                    bPartRemovedConfirmedForExchange := FALSE;

                    eOperatorExchangeState :=
                        E_OperatorExchangeState.ExchangeComplete;

                ELSE

                    // Original enabled Puck Locker sequence.
                    eOperatorExchangeState :=
                        E_OperatorExchangeState.WaitingForPuckRemoval;

                END_IF


            // -------------------------------------------------------------
            // FAIL result.
            // -------------------------------------------------------------
            ELSIF bPendingOperatorResultFail THEN

                // The rejected part must be placed at the reject sensor.
                eOperatorExchangeState :=
                    E_OperatorExchangeState.WaitingForRejectConfirmation;

            END_IF

        END_IF


    // ========================================================================
    E_OperatorExchangeState.WaitingForPuckRemoval:
    // ========================================================================

        bOperatorExchangeComplete := FALSE;


        // Recovery protection:
        //
        // If the Puck Locker is disabled while the sequence is already in
        // this state, no puck removal must be awaited.
        IF GVL_HMI.stPuckLocker.eMode =
            E_PuckLockerMode.Disabled THEN

            bPartRemovedConfirmedForExchange := FALSE;

            eOperatorExchangeState :=
                E_OperatorExchangeState.ExchangeComplete;

        ELSE

            // Once the locker accepts the release request,
            // the part-removal handshake is no longer needed.
            IF GVL_MASTER.stPuckLocker.eState =
                E_PuckLockerState.ReleasingPuck THEN

                bPartRemovedConfirmedForExchange := FALSE;

            END_IF


            // Advance when the old puck is physically gone.
            //
            // Do not require the locker to remain in ReleasingPuck.
            IF NOT GVL_MASTER.stPuckLocker.bPuckDetected THEN

                eOperatorExchangeState :=
                    E_OperatorExchangeState.WaitingForNewPuck;

            END_IF

        END_IF


    // ========================================================================
    E_OperatorExchangeState.WaitingForRejectConfirmation:
    // ========================================================================

        bOperatorExchangeComplete := FALSE;


        // Latch the reject-bin sensor pulse.
        IF rtPartPresentReject.Q THEN

            bRejectConfirmedForExchange := TRUE;

        END_IF


        // Complete the rejected-part exchange when:
        //
        // 1. The rejected part has been confirmed at the reject sensor.
        // 2. The part is no longer present in the operator nest.
        // 3. The Puck Locker is disabled, or the puck remains present
        //    and locked.
        IF bRejectConfirmedForExchange
			   AND bPartRemovedConfirmedForExchange
			   AND
			   (
                GVL_HMI.stPuckLocker.eMode =
                    E_PuckLockerMode.Disabled

                OR
                (
                    GVL_MASTER.stPuckLocker.bPuckDetected
                    AND
                    GVL_MASTER.stPuckLocker.bPuckLocked
                    AND
                    GVL_MASTER.stPuckLocker.eState =
                        E_PuckLockerState.Locked
                )
           ) THEN

            bPartRemovedConfirmedForExchange := FALSE;

            eOperatorExchangeState :=
                E_OperatorExchangeState.ExchangeComplete;

        END_IF


    // ========================================================================
    E_OperatorExchangeState.WaitingForNewPuck:
    // ========================================================================

        bOperatorExchangeComplete := FALSE;


        // Recovery protection:
        //
        // A replacement puck is not required when the locker is disabled.
        IF GVL_HMI.stPuckLocker.eMode =
            E_PuckLockerMode.Disabled THEN

            eOperatorExchangeState :=
                E_OperatorExchangeState.ExchangeComplete;


        // Original enabled Puck Locker sequence.
        ELSIF GVL_MASTER.stPuckLocker.bPuckDetected THEN

            eOperatorExchangeState :=
                E_OperatorExchangeState.WaitingForPuckLocked;

        END_IF


    // ========================================================================
    E_OperatorExchangeState.WaitingForPuckLocked:
    // ========================================================================

        bOperatorExchangeComplete := FALSE;


        // Recovery protection:
        //
        // Physical puck locking is not required when the locker is disabled.
        IF GVL_HMI.stPuckLocker.eMode =
            E_PuckLockerMode.Disabled THEN

            eOperatorExchangeState :=
                E_OperatorExchangeState.ExchangeComplete;


        // Original enabled Puck Locker sequence.
        ELSIF GVL_MASTER.stPuckLocker.bPuckDetected
           AND GVL_MASTER.stPuckLocker.bPuckLocked
           AND GVL_MASTER.stPuckLocker.eState =
                E_PuckLockerState.Locked THEN

            // Loading a new part remains optional.
            eOperatorExchangeState :=
                E_OperatorExchangeState.ExchangeComplete;

        END_IF


    // ========================================================================
    E_OperatorExchangeState.WaitingForPartLoading:
    // ========================================================================

        // Original behavior preserved.
        //
        // Require an actual OFF -> ON transition from the operator nest
        // sensor. The puck must also be present and locked.
        IF GVL_MASTER.astNestTracking[
                iOperatorNestIndex
           ].bPartLoadedPulse
           AND GVL_MASTER.stPuckLocker.bPuckDetected
           AND GVL_MASTER.stPuckLocker.bPuckLocked
           AND GVL_MASTER.stPuckLocker.eState =
                E_PuckLockerState.Locked THEN

            eOperatorExchangeState :=
                E_OperatorExchangeState.ExchangeComplete;

        END_IF


    // ========================================================================
    E_OperatorExchangeState.ExchangeComplete:
    // ========================================================================

        // Keep the index permission active until the table starts moving.
        bOperatorExchangeComplete := TRUE;


        // The previous result and its disposition are complete.
        M_ClearCompletedOperatorNestResult();


        IF GVL_MASTER.stNestTable.bNestInMotion THEN

            bPendingOperatorResultPass := FALSE;
            bPendingOperatorResultFail := FALSE;

            bPartRemovedConfirmedForExchange := FALSE;
            bRejectConfirmedForExchange := FALSE;

            eOperatorExchangeState :=
                E_OperatorExchangeState.WaitingForTableIndexComplete;

        END_IF


    // ========================================================================
    E_OperatorExchangeState.WaitingForTableIndexComplete:
    // ========================================================================

        bOperatorExchangeComplete := TRUE;


        IF eNestState = E_NestState.TESTING
           AND NOT GVL_MASTER.stNestTable.bNestInMotion
           AND GVL_MASTER.stNestTable.bNestReadySensor
           AND GVL_MASTER.stNestTable.bNestLockedSensor
           AND eCurrentNestPos <> E_NestPosition.Unknown THEN

            bOperatorExchangeComplete := FALSE;

            bPendingOperatorResultPass := FALSE;
            bPendingOperatorResultFail := FALSE;

            bPartRemovedConfirmedForExchange := FALSE;
            bRejectConfirmedForExchange := FALSE;

            eOperatorExchangeState :=
                E_OperatorExchangeState.Idle;

        END_IF


    // ========================================================================
    ELSE
    // ========================================================================

        bOperatorExchangeComplete := FALSE;

        bPendingOperatorResultPass := FALSE;
        bPendingOperatorResultFail := FALSE;

        bPartRemovedConfirmedForExchange := FALSE;
        bRejectConfirmedForExchange := FALSE;

        eOperatorExchangeState :=
            E_OperatorExchangeState.Idle;

END_CASE
END_METHOD

METHOD PRIVATE M_PreExecution : BOOL
VAR

END_VAR
// =================================================================================
// SYSTEM TIMERS
// =================================================================================
// Update initialization and safety timers on every PLC scan cycle
tonSys_Init(IN := GVL_MASTER.stMachineStatus.bInitialising);
tonSys_InitTimeout(IN := GVL_MASTER.stMachineStatus.bInitialising);

// TwinSAFE circuit stabilization timer (10 seconds)
tonSafety(IN := (GVL_MASTER.stMachineStatus.eMachineState = E_MachineState.SAFETY), PT := T#10S);

// 
//  fbStopTrigger(CLK := GVL_Master.i_bButtonStop);
//  bButtonStop := fbStopTrigger.Q;

// =================================================================================
// HMI MESSAGE CLEARING
// =================================================================================
// Clear old system messages if the machine is not actively in production
// Uses the proper ENUM namespace from your MASTER folder
IF GVL_MASTER.stMachineStatus.eMachineState <> E_MachineState.SYSTEM_AUTO_CYCLE THEN
    sMachineMessage := '';            
END_IF


// =================================================================================
// CRITICAL FAULT INTERLOCK (Watchdog)
// =================================================================================
// If Kistler hardware is NOT ready, force the state machine to FAULT immediately
// Exception: Do not override if the system is currently in SAFETY or POWER_UP
IF NOT GVL_MASTER.bKistlerSystemReady 
    AND GVL_MASTER.stMachineStatus.eMachineState <> E_MachineState.SAFETY 
    AND GVL_MASTER.stMachineStatus.eMachineState <> E_MachineState.SYSTEM_POWER_UP THEN
    
    GVL_MASTER.stMachineStatus.eMachineState := E_MachineState.FAULT;
END_IF


// =================================================================================
// START LEDs BUTTON OFF
// =================================================================================
eMode_LED_Start := E_LEDs_Mode.OFF;
eMode_LED_Reset := E_LEDs_Mode.OFF;

// =================================================================================
// METHOD EXECUTION FEEDBACK (Return True)
// =================================================================================
// Returning TRUE confirms the pre-execution routine completed successfully
M_PreExecution := TRUE;
END_METHOD

METHOD M_ProcessCycle : BOOL
VAR
bControlledStopActive 	: BOOL;
rTrigTwoHands : R_TRIG; // Edge trigger to detect single press of the two-hand safety signal

bManualIndexerOnly        : BOOL;
bManualKistlerOnly        : BOOL;
bManualIndexerAndKistler  : BOOL;



END_VAR
// Process cycle is allowed during:
//
// 1. Automatic production.
// 2. Manual Mode when the Kistler or indexer manual function is enabled.
bProcessCycleAllowed :=
    (
        GVL_MASTER.stMachineStatus.eMachineState =
            E_MachineState.SYSTEM_AUTO_CYCLE
    )
    OR
    (
        GVL_MASTER.stMachineStatus.eMachineState =
            E_MachineState.MANUAL_MODE

        AND
        (
            GVL_HMI.i_bHMIKistlerManualEnable
            OR
            GVL_HMI.i_bHMIIndexerManualEnable
        )
    );


bManualIndexerOnly :=
    GVL_HMI.i_bHMIIndexerManualEnable
    AND NOT GVL_HMI.i_bHMIKistlerManualEnable;


bManualKistlerOnly :=
    GVL_HMI.i_bHMIKistlerManualEnable
    AND NOT GVL_HMI.i_bHMIIndexerManualEnable;


bManualIndexerAndKistler :=
    GVL_HMI.i_bHMIIndexerManualEnable
    AND GVL_HMI.i_bHMIKistlerManualEnable;


// -----------------------------------------------------------------------------
// If process execution is not permitted, reset the temporary process states.
//
// Stored nest PASS/FAIL results must not be cleared by M_ResetProcessCycle.
// -----------------------------------------------------------------------------
IF NOT bProcessCycleAllowed THEN

    M_ResetProcessCycle();

    RETURN;

END_IF


// -----------------------------------------------------------------------------
// Common timers and edge detections.
// -----------------------------------------------------------------------------
rTrigTwoHands(
    CLK := GVL_IO.stSafety.bTwoHandsSafe
);


tTwoHandTargetTime :=
    REAL_TO_TIME(rHmiTwoHandPresetTime);


tTwoHandHoldTimer(
    IN := GVL_IO.stSafety.bTwoHandsSafe,
    PT := tTwoHandTargetTime
);


rtPartPresentReject(
    CLK := GVL_MASTER.stSensors.bPartPresent_Reject
);


// ============================================================================
// COMMON POSITION AND TRACKING UPDATE
//
// These methods are required in both Auto and Manual Mode.
// ============================================================================
eCurrentNestPos :=
    M_GetCurrentPosition();


M_UpdateActiveNestPositions();

M_UpdateOperatorNestTracking();


// ============================================================================
// AUTOMATIC OPERATOR EXCHANGE
//
// The following methods belong only to automatic production.
//
// They must not:
//
// - send a PASS/FAIL disposition while in Manual Mode;
// - release a puck during Manual Mode;
// - clear a completed nest result during Manual Mode;
// - block manual index movement waiting for part removal;
// - block manual index movement waiting for reject confirmation;
// - block manual index movement waiting for a puck.
// ============================================================================
IF GVL_MASTER.stMachineStatus.eMachineState =
    E_MachineState.SYSTEM_AUTO_CYCLE THEN

    M_UpdatePuckLockerPartRemovalStatus();

    M_ConfirmPuckLockerDisposition();

    M_PuckLockerDisposition();

    M_OperatorExchangeControl();

ELSE

    // Prevent a stale removal confirmation from being sent to the
    // Puck Locker while the machine is operating manually.
    GVL_MASTER.stPuckLocker.bPartRemovedFromNest := FALSE;

END_IF


// -----------------------------------------------------------------------------
// Determine whether the current physical table position is different from
// the most recently processed Kistler position.
// -----------------------------------------------------------------------------
bNestNewPositionReady :=
    (
        eCurrentNestPos <> E_NestPosition.UNKNOWN
    )
    AND
    (
        eCurrentNestPos <> eLastTestedNestPos
    );


// -----------------------------------------------------------------------------
// Capture live Kistler values while an automatic or manual sequence is active.
//
// This does not store PASS/FAIL. It only updates the live maximum values.
// -----------------------------------------------------------------------------
IF GVL_MASTER.stProcess.bKistlerCycleRequest
   AND NOT stKistlerOutTelegram.bSequenceEnd THEN

    M_HMIKistlerResult(
        eNestPosition := eCurrentNestPos,
        bPartOK       := FALSE,
        bPartNOK      := FALSE,
        rForce        := stKistler_Status.rLiveForce,
        rDistance     := stKistler_Status.rLiveDistance,
        bResetValues  := FALSE
    );

END_IF


// ============================================================================
// PROCESS CYCLE COORDINATOR
// ============================================================================
CASE GVL_MASTER.stMachineStatus.eMachineState OF


    // ========================================================================
    // AUTOMATIC CYCLE
    // ========================================================================
    E_MachineState.SYSTEM_AUTO_CYCLE:

        CASE eProcessCycleState OF


            // =================================================================
            E_ProcessCycle_State.IDLE:
            // =================================================================

                GVL_MASTER.stProcess.bKistlerCycleRequest := FALSE;
                GVL_MASTER.stProcess.bKistlerCycleDone    := FALSE;
                GVL_MASTER.stProcess.bKistlerHomeDone     := FALSE;
                GVL_MASTER.stProcess.bReleaseNestRotation := FALSE;

                tonAfterKistlerDelay(IN := FALSE);

                IF bProcessCycleAllowed THEN

                    eProcessCycleState :=
                        E_ProcessCycle_State.WAIT_NEST_TESTING_READY;

                END_IF


            // =================================================================
            E_ProcessCycle_State.WAIT_NEST_TESTING_READY:
            // =================================================================

                GVL_MASTER.stProcess.bKistlerCycleRequest := FALSE;
                GVL_MASTER.stProcess.bReleaseNestRotation := FALSE;

                tonAfterKistlerDelay(IN := FALSE);


                IF NOT bProcessCycleAllowed THEN

                    eProcessCycleState :=
                        E_ProcessCycle_State.IDLE;


                // -------------------------------------------------------------
                // Invalid table position.
                //
                // Never execute the Kistler if the PLC cannot determine which
                // physical nest is currently at the test station.
                // -------------------------------------------------------------
                ELSIF GVL_MASTER.stProcess.bNestTestingReady
                      AND eNestState = E_NestState.TESTING
                      AND eCurrentNestPos =
                            E_NestPosition.UNKNOWN THEN

                    GVL_MASTER.stProcess.bKistlerCycleRequest := FALSE;
                    GVL_MASTER.stProcess.bReleaseNestRotation := FALSE;
                    GVL_MASTER.stProcess.bKistlerCycleDone    := FALSE;
                    GVL_MASTER.stProcess.bKistlerHomeDone     := FALSE;

                    eProcessCycleState :=
                        E_ProcessCycle_State.FAULT;


                // -------------------------------------------------------------
                // Same position already processed, or no part at Kistler.
                //
                // Do not execute another Kistler cycle. Release the table.
                // -------------------------------------------------------------
                ELSIF GVL_MASTER.stProcess.bNestTestingReady
                      AND eNestState = E_NestState.TESTING
                      AND GVL_MASTER.stNestTable.bNestReadySensor
                      AND GVL_MASTER.stNestTable.bNestLockedSensor
                      AND NOT GVL_MASTER.stNestTable.bNestInMotion
                      AND eCurrentNestPos <>
                            E_NestPosition.UNKNOWN
                      AND
                      (
                          NOT bNestNewPositionReady
                          OR
                          NOT GVL_MASTER.stSensors.bPartPresent_Kistler
                      ) THEN

                    GVL_MASTER.stProcess.bKistlerCycleRequest := FALSE;
                    GVL_MASTER.stProcess.bKistlerCycleDone    := FALSE;

                    // Kistler side is considered complete because there is
                    // no valid new part to test.
                    GVL_MASTER.stProcess.bKistlerHomeDone := TRUE;


                    IF bNestNewPositionReady THEN

                        // New position without a part.
                        // Remove any previous HMI measurement result.
                        M_HMIKistlerResult(
                            eNestPosition := eCurrentNestPos,
                            bPartOK       := FALSE,
                            bPartNOK      := FALSE,
                            rForce        := 0.0,
                            rDistance     := 0.0,
                            bResetValues  := TRUE
                        );

                        eLastTestedNestPos :=
                            eCurrentNestPos;

                    END_IF


                    GVL_MASTER.stProcess.bReleaseNestRotation := TRUE;

                    eProcessCycleState :=
                        E_ProcessCycle_State.RELEASE_NEST;


                // -------------------------------------------------------------
                // New enabled nest containing a part.
                //
                // Execute the Kistler sequence.
                // -------------------------------------------------------------
                ELSIF GVL_MASTER.stProcess.bNestTestingReady
                      AND eNestState = E_NestState.TESTING
                      AND GVL_MASTER.stNestTable.bNestReadySensor
                      AND GVL_MASTER.stNestTable.bNestLockedSensor
                      AND NOT GVL_MASTER.stNestTable.bNestInMotion
                      AND stKistler_Status.eKistlerState =
                            E_KistlerState.READY
                      AND NOT stKistler_Status.bError
                      AND NOT bKistlerRecoveryHomeRequest
                      AND bNestNewPositionReady
                      AND GVL_MASTER.stSensors.bPartPresent_Kistler
                      AND M_IsNestEnabled(eCurrentNestPos) THEN

                    GVL_MASTER.stProcess.bKistlerCycleDone := FALSE;
                    GVL_MASTER.stProcess.bKistlerHomeDone  := FALSE;

                    bKistlerResultStored := FALSE;


                    // Clear the previous HMI measurement values.
                    M_HMIKistlerResult(
                        eNestPosition := eCurrentNestPos,
                        bPartOK       := FALSE,
                        bPartNOK      := FALSE,
                        rForce        := 0.0,
                        rDistance     := 0.0,
                        bResetValues  := TRUE
                    );


                    eProcessCycleState :=
                        E_ProcessCycle_State.REQUEST_KISTLER;


                // -------------------------------------------------------------
                // Nest disabled from HMI.
                //
                // Skip the Kistler test and release the table normally.
                // -------------------------------------------------------------
                ELSIF GVL_MASTER.stProcess.bNestTestingReady
                      AND eNestState = E_NestState.TESTING
                      AND GVL_MASTER.stNestTable.bNestReadySensor
                      AND GVL_MASTER.stNestTable.bNestLockedSensor
                      AND NOT GVL_MASTER.stNestTable.bNestInMotion
                      AND eCurrentNestPos <>
                            E_NestPosition.UNKNOWN
                      AND bNestNewPositionReady
                      AND GVL_MASTER.stSensors.bPartPresent_Kistler
                      AND NOT M_IsNestEnabled(eCurrentNestPos) THEN

                    GVL_MASTER.stProcess.bKistlerCycleRequest := FALSE;
                    GVL_MASTER.stProcess.bKistlerCycleDone    := FALSE;
                    GVL_MASTER.stProcess.bKistlerHomeDone     := TRUE;


                    M_HMIKistlerResult(
                        eNestPosition := eCurrentNestPos,
                        bPartOK       := FALSE,
                        bPartNOK      := FALSE,
                        rForce        := 0.0,
                        rDistance     := 0.0,
                        bResetValues  := TRUE
                    );


                    eLastTestedNestPos :=
                        eCurrentNestPos;

                    GVL_MASTER.stProcess.bReleaseNestRotation :=
                        TRUE;

                    eProcessCycleState :=
                        E_ProcessCycle_State.RELEASE_NEST;

                END_IF


            // =================================================================
            E_ProcessCycle_State.REQUEST_KISTLER:
            // =================================================================

                GVL_MASTER.stProcess.bKistlerCycleRequest := TRUE;


                IF stKistler_Status.bError THEN

                    GVL_MASTER.stProcess.bKistlerCycleRequest :=
                        FALSE;

                    eProcessCycleState :=
                        E_ProcessCycle_State.FAULT;


                ELSIF stKistler_Status.eKistlerState <>
                      E_KistlerState.READY THEN

                    eProcessCycleState :=
                        E_ProcessCycle_State.WAIT_KISTLER_DONE;

                END_IF


            // =================================================================
            E_ProcessCycle_State.WAIT_KISTLER_DONE:
            // =================================================================

                // Keep the request active while the Kistler is executing.
                GVL_MASTER.stProcess.bKistlerCycleRequest := TRUE;


                IF stKistler_Status.bError THEN

                    GVL_MASTER.stProcess.bKistlerCycleRequest :=
                        FALSE;

                    eProcessCycleState :=
                        E_ProcessCycle_State.FAULT;


                ELSIF stKistler_Status.eKistlerState =
                      E_KistlerState.DONE THEN

                    GVL_MASTER.stProcess.bKistlerCycleRequest :=
                        FALSE;

                    GVL_MASTER.stProcess.bKistlerCycleDone :=
                        TRUE;

                    eProcessCycleState :=
                        E_ProcessCycle_State.WAIT_KISTLER_HOME;

                END_IF


            // =================================================================
            E_ProcessCycle_State.WAIT_KISTLER_HOME:
            // =================================================================

                M_StoreKistlerResult();

                GVL_MASTER.stProcess.bKistlerCycleRequest := FALSE;


                IF stKistler_Status.bError THEN

                    eProcessCycleState :=
                        E_ProcessCycle_State.FAULT;


                ELSIF stKistlerOutTelegram.bHomePosReached
                      OR stKistlerOutTelegram.bRefPosReached
                      OR stKistler_Status.bInPosition THEN

                    GVL_MASTER.test :=
                        GVL_MASTER.test + 1;

                    GVL_MASTER.stProcess.bKistlerHomeDone :=
                        TRUE;

                    GVL_MASTER.stProcess.bKistlerCycleDone :=
                        TRUE;


                    // ---------------------------------------------------------
                    // Store the process result.
                    // ---------------------------------------------------------
                    IF stKistler_Status.bPartOK THEN

                        GVL_MASTER.stProcess.bKistlerResultOK :=
                            TRUE;

                        GVL_MASTER.stProcess.bKistlerResultNOK :=
                            FALSE;


                    ELSIF stKistler_Status.bPartNOK THEN

                        GVL_MASTER.stProcess.bKistlerResultOK :=
                            FALSE;

                        GVL_MASTER.stProcess.bKistlerResultNOK :=
                            TRUE;


                    ELSE

                        // Test ended without a valid OK/NOK result.
                        // Preserve the existing behavior.
                        RETURN;

                    END_IF


                    eLastTestedNestPos :=
                        eCurrentNestPos;


                    IF NOT M_HMIKistlerResult(
                        eNestPosition := eCurrentNestPos,
                        bPartOK       := stKistler_Status.bPartOK,
                        bPartNOK      := stKistler_Status.bPartNOK,
                        rForce        := stKistler_Status.rLiveForce,
                        rDistance     := stKistler_Status.rLiveDistance,
                        bResetValues  := FALSE
                    ) THEN

                        RETURN;

                    END_IF


                    eProcessCycleState :=
                        E_ProcessCycle_State.WAIT_AFTER_KISTLER;

                END_IF


            // =================================================================
            E_ProcessCycle_State.WAIT_AFTER_KISTLER:
            // =================================================================

                IF stKistlerOutTelegram.bSequenceEnd
                   AND
                   (
                       stKistlerOutTelegram.bHomePosReached
                       OR
                       stKistlerOutTelegram.bRefPosReached
                       OR
                       stKistler_Status.bInPosition
                   ) THEN

                    GVL_MASTER.stProcess.bReleaseNestRotation :=
                        TRUE;

                    eProcessCycleState :=
                        E_ProcessCycle_State.RELEASE_NEST;

                END_IF


            // =================================================================
            E_ProcessCycle_State.RELEASE_NEST:
            // =================================================================

                // Keep the release request active until NestTableControl
                // consumes it.
                GVL_MASTER.stProcess.bReleaseNestRotation := TRUE;


                IF eNestState <> E_NestState.TESTING
                   OR NOT GVL_MASTER.stProcess.bNestTestingReady THEN

                    GVL_MASTER.stProcess.bReleaseNestRotation :=
                        FALSE;

                    GVL_MASTER.stProcess.bKistlerCycleRequest :=
                        FALSE;

                    GVL_MASTER.stProcess.bKistlerCycleDone :=
                        FALSE;

                    GVL_MASTER.stProcess.bKistlerHomeDone :=
                        FALSE;

                    tonAfterKistlerDelay(IN := FALSE);


                    eProcessCycleState :=
                        E_ProcessCycle_State.WAIT_NEST_TESTING_READY;

                END_IF


            // =================================================================
            E_ProcessCycle_State.FAULT:
            // =================================================================

                GVL_MASTER.stProcess.bKistlerCycleRequest := FALSE;
                GVL_MASTER.stProcess.bReleaseNestRotation := FALSE;

                tonAfterKistlerDelay(IN := FALSE);

                M_ResetProcessCycle();

                GVL_MASTER.stMachineStatus.eMachineState :=
                    E_MachineState.FAULT;


                IF GVL_MASTER.stMachineStatus.bStopped THEN

                    eProcessCycleState :=
                        E_ProcessCycle_State.IDLE;

                END_IF


            // =================================================================
            ELSE
            // =================================================================

                eProcessCycleState :=
                    E_ProcessCycle_State.IDLE;

        END_CASE


    // ========================================================================
    // MANUAL MODE
    // ========================================================================
    E_MachineState.MANUAL_MODE:

        CASE eProcessCycleState OF


            // =================================================================
            E_ProcessCycle_State.IDLE:
            // =================================================================

                GVL_MASTER.stProcess.bKistlerCycleRequest := FALSE;
                GVL_MASTER.stProcess.bKistlerCycleDone    := FALSE;
                GVL_MASTER.stProcess.bKistlerHomeDone     := FALSE;
                GVL_MASTER.stProcess.bReleaseNestRotation := FALSE;

                GVL_MASTER.stProcess.bKistlerResultOK  := FALSE;
                GVL_MASTER.stProcess.bKistlerResultNOK := FALSE;

                tonAfterKistlerDelay(IN := FALSE);


                IF bManualIndexerOnly
                   OR bManualIndexerAndKistler THEN

                    eProcessCycleState :=
                        E_ProcessCycle_State.WAIT_NEST_TESTING_READY;


                ELSIF bManualKistlerOnly
                      AND NOT GVL_MASTER.stProcess.bNestTestingReady
                      AND stKistler_Status.eKistlerState =
                            E_KistlerState.READY
                      AND NOT stKistler_Status.bError
                      AND NOT bKistlerRecoveryHomeRequest THEN

                    GVL_MASTER.stProcess.bNestTestingReady :=
                        FALSE;

                    eProcessCycleState :=
                        E_ProcessCycle_State.REQUEST_KISTLER;

                END_IF


            // =================================================================
            E_ProcessCycle_State.WAIT_NEST_TESTING_READY:
            // =================================================================

                GVL_MASTER.stProcess.bKistlerCycleRequest := FALSE;
                GVL_MASTER.stProcess.bReleaseNestRotation := FALSE;

                tonAfterKistlerDelay(IN := FALSE);


                IF NOT (
                    bManualIndexerOnly
                    OR bManualIndexerAndKistler
                ) THEN

                    eProcessCycleState :=
                        E_ProcessCycle_State.IDLE;


                ELSIF GVL_MASTER.stProcess.bNestTestingReady
                      AND eNestState = E_NestState.TESTING
                      AND bManualIndexerAndKistler
                      AND stKistler_Status.eKistlerState =
                            E_KistlerState.READY
                      AND NOT stKistler_Status.bError
                      AND NOT bKistlerRecoveryHomeRequest THEN

                    eProcessCycleState :=
                        E_ProcessCycle_State.REQUEST_KISTLER;


                ELSIF GVL_MASTER.stProcess.bNestTestingReady
                      AND eNestState = E_NestState.TESTING
                      AND bManualIndexerOnly THEN

                    GVL_MASTER.stProcess.bKistlerCycleRequest :=
                        FALSE;

                    GVL_MASTER.stProcess.bKistlerHomeDone :=
                        TRUE;

                    GVL_MASTER.stProcess.bReleaseNestRotation :=
                        TRUE;

                    eProcessCycleState :=
                        E_ProcessCycle_State.RELEASE_NEST;

                END_IF


            // =================================================================
            E_ProcessCycle_State.REQUEST_KISTLER:
            // =================================================================

                // Kistler already reacted.
                IF stKistler_Status.eKistlerState <>
                    E_KistlerState.READY THEN

                    eProcessCycleState :=
                        E_ProcessCycle_State.WAIT_KISTLER_DONE;


                // -------------------------------------------------------------
                // Manual Kistler only.
                //
                // Start only on the two-hand rising edge.
                // -------------------------------------------------------------
                ELSIF bManualKistlerOnly
                      AND GVL_IO.stSafety.bSafetyOK
                      AND rTrigTwoHands.Q
                      AND GVL_MASTER.stNestTable.bNestReadySensor
                      AND GVL_MASTER.stNestTable.bNestLockedSensor
                      AND NOT stKistler_Status.bError
                      AND NOT bKistlerRecoveryHomeRequest THEN

                    GVL_MASTER.stProcess.bKistlerCycleRequest :=
                        TRUE;


                // -------------------------------------------------------------
                // Manual indexer and Kistler.
                // -------------------------------------------------------------
                ELSIF bManualIndexerAndKistler
                      AND GVL_MASTER.stProcess.bNestTestingReady
                      AND eNestState = E_NestState.TESTING
                      AND GVL_MASTER.stNestTable.bNestReadySensor
                      AND GVL_MASTER.stNestTable.bNestLockedSensor
                      AND NOT GVL_MASTER.stNestTable.bNestInMotion
                      AND eCurrentNestPos <>
                            E_NestPosition.UNKNOWN
                      AND bNestNewPositionReady
                      AND NOT stKistler_Status.bError
                      AND NOT bKistlerRecoveryHomeRequest THEN

                    GVL_MASTER.stProcess.bKistlerCycleRequest :=
                        TRUE;


                ELSIF stKistler_Status.bError THEN

                    GVL_MASTER.stProcess.bKistlerCycleRequest :=
                        FALSE;

                    eProcessCycleState :=
                        E_ProcessCycle_State.FAULT;

                END_IF


            // =================================================================
            E_ProcessCycle_State.WAIT_KISTLER_DONE:
            // =================================================================

                GVL_MASTER.stProcess.bKistlerCycleRequest := TRUE;


                IF stKistler_Status.bError THEN

                    GVL_MASTER.stProcess.bKistlerCycleRequest :=
                        FALSE;

                    eProcessCycleState :=
                        E_ProcessCycle_State.FAULT;


                ELSIF stKistler_Status.eKistlerState =
                      E_KistlerState.DONE THEN

                    // Capture the final available measurements.
                    M_HMIKistlerResult(
                        eNestPosition := eCurrentNestPos,
                        bPartOK       := FALSE,
                        bPartNOK      := FALSE,
                        rForce        := stKistler_Status.rLiveForce,
                        rDistance     := stKistler_Status.rLiveDistance,
                        bResetValues  := FALSE
                    );


                    GVL_MASTER.stProcess.bKistlerCycleRequest :=
                        FALSE;

                    GVL_MASTER.stProcess.bKistlerCycleDone :=
                        TRUE;


                    IF bManualIndexerAndKistler THEN

                        eLastTestedNestPos :=
                            eCurrentNestPos;

                        eProcessCycleState :=
                            E_ProcessCycle_State.WAIT_KISTLER_HOME;

                    ELSE

                        eProcessCycleState :=
                            E_ProcessCycle_State.IDLE;

                    END_IF

                END_IF


            // =================================================================
            E_ProcessCycle_State.WAIT_KISTLER_HOME:
            // =================================================================

                GVL_MASTER.stProcess.bKistlerCycleRequest := FALSE;


                IF stKistler_Status.bError THEN

                    eProcessCycleState :=
                        E_ProcessCycle_State.FAULT;


                ELSIF stKistlerOutTelegram.bHomePosReached
                      OR stKistlerOutTelegram.bRefPosReached
                      OR stKistler_Status.bInPosition THEN

                    GVL_MASTER.stProcess.bKistlerHomeDone :=
                        TRUE;


                    IF bManualIndexerAndKistler THEN

                        eProcessCycleState :=
                            E_ProcessCycle_State.WAIT_AFTER_KISTLER;

                    ELSE

                        eProcessCycleState :=
                            E_ProcessCycle_State.IDLE;

                    END_IF

                END_IF


            // =================================================================
            E_ProcessCycle_State.WAIT_AFTER_KISTLER:
            // =================================================================

                IF stKistlerOutTelegram.bSequenceEnd
                   AND
                   (
                       stKistlerOutTelegram.bHomePosReached
                       OR
                       stKistlerOutTelegram.bRefPosReached
                       OR
                       stKistler_Status.bInPosition
                   ) THEN

                    GVL_MASTER.stProcess.bReleaseNestRotation :=
                        TRUE;

                    eProcessCycleState :=
                        E_ProcessCycle_State.RELEASE_NEST;

                END_IF


            // =================================================================
            E_ProcessCycle_State.RELEASE_NEST:
            // =================================================================

                GVL_MASTER.stProcess.bReleaseNestRotation :=
                    TRUE;


                IF eNestState <> E_NestState.TESTING
                   OR NOT GVL_MASTER.stProcess.bNestTestingReady THEN

                    GVL_MASTER.stProcess.bReleaseNestRotation :=
                        FALSE;

                    GVL_MASTER.stProcess.bKistlerCycleRequest :=
                        FALSE;

                    GVL_MASTER.stProcess.bKistlerCycleDone :=
                        FALSE;

                    GVL_MASTER.stProcess.bKistlerHomeDone :=
                        FALSE;

                    tonAfterKistlerDelay(IN := FALSE);


                    IF bManualIndexerOnly
                       OR bManualIndexerAndKistler THEN

                        eProcessCycleState :=
                            E_ProcessCycle_State.WAIT_NEST_TESTING_READY;

                    ELSE

                        eProcessCycleState :=
                            E_ProcessCycle_State.IDLE;

                    END_IF

                END_IF


            // =================================================================
            E_ProcessCycle_State.FAULT:
            // =================================================================

                GVL_MASTER.stProcess.bKistlerCycleRequest :=
                    FALSE;

                GVL_MASTER.stProcess.bReleaseNestRotation :=
                    FALSE;

                tonAfterKistlerDelay(IN := FALSE);

                M_ResetProcessCycle();

                GVL_MASTER.stMachineStatus.eMachineState :=
                    E_MachineState.FAULT;


            // =================================================================
            ELSE
            // =================================================================

                eProcessCycleState :=
                    E_ProcessCycle_State.IDLE;

        END_CASE


    // ========================================================================
    ELSE
    // ========================================================================

        // This should normally be handled by bProcessCycleAllowed at the
        // beginning of the method.
        M_ResetProcessCycle();

END_CASE


M_ProcessCycle := TRUE;
END_METHOD

METHOD PRIVATE M_PuckLockerDisposition
VAR
	iOperatorNestIndex : INT;
    bResultPass        : BOOL;
    bResultFail        : BOOL;
END_VAR
// -----------------------------------------------------------------------------
// The operator nest must be known.
// -----------------------------------------------------------------------------
IF eOperatorNestPosition = E_NestPosition.Unknown THEN
    RETURN;
END_IF


// Process the operator disposition whenever the table is stationary,
// mechanically locked and accessible to the operator.
//
// TESTING:
//     Normal production flow.
//
// WAIT_OPERATOR_EXCHANGE:
//     Normal exchange after a completed test.
//
// IDLE:
//     Recovery flow after FAULT, STOPPED or reinitialisation.
IF (
        eNestState <> E_NestState.IDLE
        AND eNestState <> E_NestState.TESTING
        AND eNestState <> E_NestState.WAIT_OPERATOR_EXCHANGE
   )
   OR GVL_MASTER.stNestTable.bNestInMotion
   OR NOT GVL_MASTER.stNestTable.bNestReadySensor
   OR NOT GVL_MASTER.stNestTable.bNestLockedSensor
   OR eCurrentNestPos = E_NestPosition.Unknown THEN

    RETURN;

END_IF


// -----------------------------------------------------------------------------
// E_NestPosition values correspond directly to array indexes 1..4.
// -----------------------------------------------------------------------------
iOperatorNestIndex := TO_INT(eOperatorNestPosition);

IF (iOperatorNestIndex < 1) OR (iOperatorNestIndex > 4) THEN
    RETURN;
END_IF


// -----------------------------------------------------------------------------
// The nest currently accessible to the operator must contain a valid result.
// -----------------------------------------------------------------------------
IF NOT GVL_MASTER.astNestProcessResult[iOperatorNestIndex].bResultValid THEN
    RETURN;
END_IF


// -----------------------------------------------------------------------------
// Do not process the same nest disposition more than once.
// -----------------------------------------------------------------------------
IF GVL_MASTER.astNestProcessResult[iOperatorNestIndex].bDispositionSent THEN
    RETURN;
END_IF


// -----------------------------------------------------------------------------
// Copy the result locally for validation and readability.
// -----------------------------------------------------------------------------
bResultPass :=
    GVL_MASTER.astNestProcessResult[iOperatorNestIndex].bPass;

bResultFail :=
    GVL_MASTER.astNestProcessResult[iOperatorNestIndex].bFail;


// -----------------------------------------------------------------------------
// The result must contain exactly one disposition.
//
// Invalid combinations:
//     PASS = FALSE and FAIL = FALSE
//     PASS = TRUE  and FAIL = TRUE
// -----------------------------------------------------------------------------
IF bResultPass = bResultFail THEN
    RETURN;
END_IF


// -----------------------------------------------------------------------------
// PUCK LOCKER DISABLED:
//
// There is no physical locker handshake to perform.
//
// Mark the disposition as delivered internally so that the operator exchange
// sequence can continue using the normal PASS/FAIL result.
//
// FAIL still requires:
//     1. Part removal from the operator nest.
//     2. Confirmation from the reject-bin sensor.
//
// No puck presence or puck locked condition is required.
// -----------------------------------------------------------------------------
IF GVL_HMI.stPuckLocker.eMode = E_PuckLockerMode.Disabled THEN

    GVL_MASTER.astNestProcessResult[
        iOperatorNestIndex
    ].bDispositionSent := TRUE;

    RETURN;

END_IF


// -----------------------------------------------------------------------------
// A previous disposition was already sent and is still waiting for confirmation
// from PRG_PuckLocker.
// -----------------------------------------------------------------------------
IF ePendingPuckDispositionNest <> E_NestPosition.Unknown THEN
    RETURN;
END_IF


// -----------------------------------------------------------------------------
// Do not overwrite a disposition that has not yet been consumed by the locker.
// -----------------------------------------------------------------------------
IF GVL_MASTER.stPuckLocker.bApplyDisposition
   OR GVL_MASTER.stPuckLocker.bDispositionPending THEN

    RETURN;

END_IF


// -----------------------------------------------------------------------------
// PASS:
// Authorise the release of one puck.
// -----------------------------------------------------------------------------
IF bResultPass THEN

    GVL_MASTER.stPuckLocker.nRequestedRelease := 1;
    GVL_MASTER.stPuckLocker.nRequestedRemoval := 0;

    // Store the nest that originated this request so that the confirmation
    // remains associated with the correct nest even if the table moves later.
    ePendingPuckDispositionNest :=
        eOperatorNestPosition;

    // Apply the request only after all associated data has been prepared.
    GVL_MASTER.stPuckLocker.bApplyDisposition := TRUE;


// -----------------------------------------------------------------------------
// FAIL:
// Inform the locker of the rejected result, but do not authorise puck release.
// The puck must remain locked until a future PASS result is received.
// -----------------------------------------------------------------------------
ELSIF bResultFail THEN

    GVL_MASTER.stPuckLocker.nRequestedRelease := 0;
    GVL_MASTER.stPuckLocker.nRequestedRemoval := 1;

    ePendingPuckDispositionNest :=
        eOperatorNestPosition;

    // Apply the request only after all associated data has been prepared.
    GVL_MASTER.stPuckLocker.bApplyDisposition := TRUE;

END_IF
END_METHOD

METHOD PRIVATE M_ResetProcessCycle : BOOL
VAR_INPUT

END_VAR

M_ResetProcessCycle := FALSE;

eProcessCycleState := E_ProcessCycle_State.IDLE;


// =========================================================
// RESET PROCESS FLAGS
// =========================================================

GVL_MASTER.stProcess.bKistlerCycleRequest := FALSE;
GVL_MASTER.stProcess.bKistlerCycleDone := FALSE;
GVL_MASTER.stProcess.bKistlerHomeDone := FALSE;
GVL_MASTER.stProcess.bNestTestingReady := FALSE;
GVL_MASTER.stProcess.bReleaseNestRotation := FALSE;
GVL_MASTER.stProcess.bKistlerResultOK := FALSE;
GVL_MASTER.stProcess.bKistlerResultNOK := FALSE;


// =========================================================
// RESET PROCESS TIMERS
// =========================================================

tonGuideCylinderDelay(IN := FALSE);
tonGuideCylinderRetractDelay(IN := FALSE);
tonAfterKistlerDelay(IN := FALSE);


// =========================================================
// RESET ACTUATOR REQUESTS
// =========================================================

GVL_MASTER.stActuators.bGuideCylinderExtendRequest := FALSE;

GVL_MASTER.stNestTable.bSupportExtendRequest := FALSE;
GVL_MASTER.stNestTable.bSupportRetractRequest := TRUE;


// =========================================================
// RESET HMI MANUAL COMMANDS
// =========================================================

GVL_HMI.i_bHMIManualModeRequest := FALSE;
GVL_HMI.i_bHMIIndexerManualEnable := FALSE;
GVL_HMI.i_bHMIKistlerManualEnable := FALSE;


// =========================================================
// RESET KISTLER SEQUENCE COMMANDS
// =========================================================

stKistler_CMD.bStart := FALSE;
stKistler_CMD.bRunSequence := FALSE;
stKistler_CMD.bDriveToHome := FALSE;
stKistler_CMD.bDriveToRef := FALSE;
stKistler_CMD.bContinueFromWait := FALSE;
stKistler_CMD.bTareY := FALSE;


// =========================================================
// START RESET PULSE
// =========================================================

// Start the pulse only on the first execution
IF NOT bKistlerResetPulse AND NOT tonKistlerReset.Q THEN
    bKistlerResetPulse := TRUE;
END_IF;


// Reset/Acknowledge command sent to the Kistler
stKistler_CMD.bReset := bKistlerResetPulse;


// Do not send Abort at the same time as Reset
stKistler_CMD.bAbort := NOT bKistlerResetPulse;


// =========================================================
// RESET PULSE TIMER
// =========================================================

tonKistlerReset(
    IN := bKistlerResetPulse,
    PT := T#500MS
);


// =========================================================
// RESET ROUTINE COMPLETE
// =========================================================

IF tonKistlerReset.Q THEN

    // End pulse commands
    bKistlerResetPulse := FALSE;

    stKistler_CMD.bReset := FALSE;
    stKistler_CMD.bAbort := FALSE;

    // Reset the timer for the next fault/reset
    tonKistlerReset(IN := FALSE);

    // Request recovery movement on the next initialization
    bKistlerRecoveryHomeRequest := TRUE;

    // Inform caller that the reset routine is complete
    M_ResetProcessCycle := TRUE;

END_IF;
END_METHOD

METHOD PRIVATE M_StatusMapping : BOOL
VAR_INPUT



END_VAR

// =================================================================================
// KISTLER TO GLOBAL STATUS MAPPING
// =================================================================================
// Link the software/hardware safety loop to the machine status structure
GVL_MASTER.stMachineStatus.bSafety := GVL_IO.stSafety.bSystemSafeOK;

// Map the local Kistler hardware ready flag to our main control variable
bKistlerReady := stKistler_Status.bReady;

// Update the global machine fault status if the Kistler press enters an error state
IF stKistler_Status.bError THEN
	GVL_MASTER.stMachineStatus.bFault := TRUE;
END_IF

// =================================================================================
// HMI / PANEL LAMP SIGNALLING MANAGEMENT
// =================================================================================
// Control the Start Button Lamp feedback based on machine state
IF GVL_MASTER.stMachineStatus.eMachineState = E_MachineState.STOPPED AND bKistlerReady THEN
    GVL_MASTER.bStartButtonLamp := GVL_MASTER.bBlink_1Hz; // Uses standard 1Hz global clock bit
ELSIF GVL_MASTER.stMachineStatus.eMachineState = E_MachineState.SYSTEM_AUTO_CYCLE THEN
    GVL_MASTER.bStartButtonLamp := TRUE;
ELSE
    GVL_MASTER.bStartButtonLamp := FALSE;
END_IF
// =================================================================================
// METHOD EXECUTION FEEDBACK (Return True)
// =================================================================================
// Returning TRUE confirms that the status mapping routine executed successfully
M_StatusMapping := TRUE;
END_METHOD

METHOD M_StoreKistlerResult
VAR
	iNestIndex : INT;
END_VAR
IF eKistlerNestPosition = E_NestPosition.Unknown THEN
    RETURN;
END_IF;

iNestIndex := eKistlerNestPosition;

IF (iNestIndex < 1) OR (iNestIndex > 4) THEN
    RETURN;
END_IF;

// Prevent writing the same result repeatedly for several PLC scans.
IF bKistlerResultStored THEN
    RETURN;
END_IF;

IF stKistler_Status.bPartOK THEN

    GVL_MASTER.astNestProcessResult[iNestIndex].bResultValid := TRUE;
    GVL_MASTER.astNestProcessResult[iNestIndex].bPass := TRUE;
    GVL_MASTER.astNestProcessResult[iNestIndex].bFail := FALSE;
    GVL_MASTER.astNestProcessResult[iNestIndex].bDispositionSent := FALSE;

    bKistlerResultStored := TRUE;

ELSIF stKistler_Status.bPartNOK THEN

    GVL_MASTER.astNestProcessResult[iNestIndex].bResultValid := TRUE;
    GVL_MASTER.astNestProcessResult[iNestIndex].bPass := FALSE;
    GVL_MASTER.astNestProcessResult[iNestIndex].bFail := TRUE;
    GVL_MASTER.astNestProcessResult[iNestIndex].bDispositionSent := FALSE;

    bKistlerResultStored := TRUE;

END_IF;
END_METHOD

METHOD M_SupportControl
VAR_INPUT
    bExtendRequest  : BOOL; // Request to lift support
    bRetractRequest : BOOL; // Request to lower support
END_VAR
// =================================================================
// SUPPORT CYLINDER CONTROL
// =================================================================
// This method is responsible only for the support cylinder outputs.
// It does not decide Auto Cycle or Manual Mode.
// The request must come from M_ProcessCycle, M_NestTableControl,
// or later from the Kistler coordination logic.

// Safety priority: never command both coils at the same time.
IF bExtendRequest AND NOT bRetractRequest THEN

    // Lift support
    GVL_MASTER.stNestTable.qSupportExtend  := TRUE;
    GVL_MASTER.stNestTable.qSupportRetract := FALSE;


ELSIF bRetractRequest AND NOT bExtendRequest THEN

    // Lower support
    GVL_MASTER.stNestTable.qSupportExtend  := FALSE;
    GVL_MASTER.stNestTable.qSupportRetract := TRUE;



ELSE

    // No request or conflicting request:
    // keep both outputs off to avoid fighting the pneumatic valve.
    GVL_MASTER.stNestTable.qSupportExtend  := FALSE;
    GVL_MASTER.stNestTable.qSupportRetract := FALSE;



END_IF
END_METHOD

METHOD PRIVATE M_UpdateActiveNestPositions
VAR_INPUT
END_VAR
eKistlerNestPosition := eCurrentNestPos;

eOperatorNestPosition := F_GetOppositeNestPosition( eKistlerPosition := eKistlerNestPosition );

IF eKistlerNestPosition <> E_NestPosition.Unknown THEN

    iKistlerNestIndex := TO_INT(eKistlerNestPosition);

ELSE

    iKistlerNestIndex := 0;

END_IF;

IF eOperatorNestPosition <> E_NestPosition.Unknown THEN

    iOperatorNestIndex := TO_INT(eOperatorNestPosition);

ELSE

    iOperatorNestIndex := 0;

END_IF;
END_METHOD

METHOD PRIVATE M_UpdateOperatorInstruction
VAR_INPUT
END_VAR
END_METHOD

METHOD PRIVATE M_UpdateOperatorNestTracking
VAR
	iOperatorNestIndex 	: INT;
    iNest               : INT;
    bPartPresent        : BOOL;
END_VAR
// Pulses are valid for one PLC scan only.
// Clear all previous events before evaluating the current operator nest.
FOR iNest := 1 TO 4 DO

    GVL_MASTER.astNestTracking[iNest].bPartRemovedPulse := FALSE;
    GVL_MASTER.astNestTracking[iNest].bPartLoadedPulse := FALSE;

END_FOR

// Track the operator sensor while the table is safely stationary.
// IDLE is required for the initial loading sequence.
// TESTING is required for the normal unload/reload sequence.
IF (
        eNestState <> E_NestState.IDLE
        AND eNestState <> E_NestState.TESTING
        AND eNestState <> E_NestState.WAIT_OPERATOR_EXCHANGE
   )
   OR GVL_MASTER.stNestTable.bNestInMotion
   OR NOT GVL_MASTER.stNestTable.bNestReadySensor
   OR NOT GVL_MASTER.stNestTable.bNestLockedSensor
   OR eOperatorNestPosition = E_NestPosition.Unknown THEN

    RETURN;

END_IF

// E_NestPosition corresponds to indexes 1..4.
iOperatorNestIndex := TO_INT(eOperatorNestPosition);

IF (iOperatorNestIndex < 1) OR (iOperatorNestIndex > 4) THEN
    RETURN;
END_IF

// The physical sensor represents the nest currently accessible
// to the operator.
bPartPresent := GVL_MASTER.stSensors.bPartPresent_NEST;

// Detect processed part removal.
GVL_MASTER.astNestTracking[iOperatorNestIndex].bPartRemovedPulse := GVL_MASTER.astNestTracking[iOperatorNestIndex].bPreviousSensor AND NOT bPartPresent;

// Detect new part loading.
GVL_MASTER.astNestTracking[iOperatorNestIndex].bPartLoadedPulse := NOT GVL_MASTER.astNestTracking[iOperatorNestIndex].bPreviousSensor AND bPartPresent;

// Store the current occupancy status.
GVL_MASTER.astNestTracking[iOperatorNestIndex].bPartLoaded := bPartPresent;

// Save the current sensor state for the next scan.
GVL_MASTER.astNestTracking[iOperatorNestIndex].bPreviousSensor := bPartPresent;
END_METHOD

METHOD PRIVATE M_UpdatePuckLockerPartRemovalStatus
VAR
	iOperatorNestIndex : INT;
END_VAR
// Keep the removal confirmation active until the Puck Locker
// acknowledges it by leaving the Locked state.
//
// Do not forward the one-scan physical sensor pulse directly.
GVL_MASTER.stPuckLocker.bPartRemovedFromNest := bPendingOperatorResultPass AND bPartRemovedConfirmedForExchange;
END_METHOD

METHOD PRIVATE M_UpdatePuckLockerPermissives
VAR_INPUT
END_VAR
// Puck Locker is considered permissive when disabled,
// or when enabled without any latched locker fault.
GVL_MASTER.stPuckLocker.bMachinePermissive :=
    (GVL_HMI.stPuckLocker.eMode = E_PuckLockerMode.Disabled)
    OR (
        NOT GVL_MASTER.stPuckLocker.bUnexpectedRemovalFault
        AND NOT GVL_MASTER.stPuckLocker.bPuckSensorMismatch
        AND GVL_MASTER.stPuckLocker.eState <>
            E_PuckLockerState.UnexpectedPuckRemovalFault
    );


// Index movement always depends on completion of the operator exchange.
//
// When the Puck Locker is disabled, its physical sensors and locker faults
// are bypassed through bMachinePermissive, but the operator must still:
//
//     1. Remove the processed part from the nest.
//     2. Place a failed part in the reject sensor.
//     3. Complete the operator exchange sequence.
//
// The Unknown-position exception is retained for initialisation/recovery.
GVL_MASTER.stPuckLocker.bIndexPermissive :=
    GVL_MASTER.stPuckLocker.bMachinePermissive
    AND (
        bOperatorExchangeComplete
        OR eCurrentNestPos = E_NestPosition.Unknown
    );
END_METHOD

END_PROGRAM

(* stored: Version 1.1.0.1
   POU PRG_MachineControl: Id {73cce6c0-0336-454e-b089-fed285c9fc85}, SpecialFunc None
   Folder GuideCylinder: Id {f10faf9c-65dc-4eb4-9dd1-2b0b5aecf204}
   Folder Kistler: Id {9e17cfcd-c98c-45cb-bd0b-324e8c0aff3a}
   Folder Nest_Table: Id {b7ca633f-afa1-44ec-8055-793fa5c0679e}
   Folder Pick_Locker: Id {df051fcd-8c9f-4620-b035-4bdfd7cf7977}
   Folder SupportElevator: Id {7f702417-a10d-4779-8751-86ff4b21f60e}
   Method M_ClearCompletedOperatorNestResult: Id {01b8ae27-8d16-43ef-a386-7432c49082ed}
   Method M_ClearRemovedOperatorNestResult: Id {c718cf76-b546-4927-a46e-0e5025b89a81}
   Method M_ConfirmPuckLockerDisposition: Id {10b0db97-52e9-4e62-9b4d-4520c43ca38e}
   Method M_GetCurrentPosition: Id {5ad458d2-2562-4615-8d3c-a8c74f1cf84a}
   Method M_GuideCylinderControl: Id {104c92f2-fa5c-4064-a20d-a8f4a2c78ac7}
   Method M_HMIKistlerResult: Id {5ec231b7-f8ff-4c60-8cb2-2f6710f94bba}
   Method M_IsNestEnabled: Id {c565a59a-4a72-4ce9-ac82-a7eafb09ab56}
   Method M_KistlerCommandMapping: Id {5cfa21d9-3cc5-49b3-924c-97638c44a598}
   Method M_KistlerConfig_Input: Id {14c376fa-cf59-47d0-a1ae-92a997aeb833}
   Method M_KistlerConfig_Output: Id {8ae5f917-1437-4f6b-8e62-9b5bec1a92a3}
   Method M_KistlerControl: Id {142f0c7b-5ff7-4bb2-a407-a7b85664501f}
   Method M_KistlerStateMachine: Id {537fbedf-c4eb-4029-b5fd-b3d3431bc3e9}
   Method M_LEDsButtons: Id {a6680c49-408d-47a5-bfa3-499d1bfac7ad}
   Method M_NestTableControl: Id {73045679-2a70-4e2a-a7bb-96539b2fce6a}
   Method M_OperatorExchangeControl: Id {531cdfdc-4414-409e-a0f2-21c7605d741a}
   Method M_PreExecution: Id {d5c5735d-f733-481f-9f83-00134f7ccc98}
   Method M_ProcessCycle: Id {e01c53ef-c471-4f56-958b-74875adab0b2}
   Method M_PuckLockerDisposition: Id {ad617b9e-72f0-4e71-8779-255d6dead4ac}
   Method M_ResetProcessCycle: Id {454cd463-1fae-4730-b15d-6fd1047cb008}
   Method M_StatusMapping: Id {e76387c3-2b6b-4ab8-8e2c-031286cbd112}
   Method M_StoreKistlerResult: Id {44a9f0cc-607f-440e-a240-216b02f970e5}
   Method M_SupportControl: Id {64d76664-69d4-4214-9755-744a37e12132}
   Method M_UpdateActiveNestPositions: Id {a175beaf-3ad8-4d7b-8c4f-5074246f2c65}
   Method M_UpdateOperatorInstruction: Id {9003e453-721d-4c1e-a060-193bc77fe83e}
   Method M_UpdateOperatorNestTracking: Id {d4e87f72-d62a-4a59-bdf7-747a3fa48afb}
   Method M_UpdatePuckLockerPartRemovalStatus: Id {f9bf3ed2-647f-49ac-acef-7d7719e93b2e}
   Method M_UpdatePuckLockerPermissives: Id {a5082c5a-ff24-4e5c-a334-ef2912094065} *)
